(* CODESYS project TestComClose.project

Project tree, tasks and I/O mapping:
  XV100 : XV100, Eaton Automation, version 3.5.3.0
    application Application
      libraries: Standard, 3.5.2.0 (System); TSR Libary, 0.95 (Eaton Automation)
      task Task (cyclic, interval t#10ms, priority 1) calls MAIN
      program MAIN [ST]
*)

// XV100/Application/MAIN
PROGRAM MAIN
VAR
	Execute					:BOOL;				//Startbedingung für den FB.
	Com						:INT;				//Die Nummer des Com Ports.
	SendData				:STRING;			//Der String der Gesendet werden soll.
	Port					:BOOL;				//Wenn = 0 Wird der Port geschlossen, Wenn = 1 Wird der Port geöffnet.
												//FB Ausgänge
	Busy					:BOOL;				//Das Busy bit.
	Done					:BOOL;				//Ist 1 wenn FB fertig ist.
	ReceivedData			:STRING;			//Der Empfangene Daten String.
	State					:WORD;				//Der ENUM Wert für die ENUM Tabelle.
	Error					:BOOL;				//Ist 1 wenn es einen Error gab.	
	TLfb_COM						:TSR_Com;
END_VAR

TLfb_COM(
	xExecute:=Execute , 
	iCom:=Com , 
	stSendData:=SendData , 
	xPort:=Port , 
	xBusy=>Busy , 
	xDone=>Done , 
	stReceivedData=>ReceivedData , 
	wState=>State , 
	xError=>Error );

END_PROGRAM
